TYPE AlbertsSettings EXTENDS TcoData.Entity :
STRUCT
	ServoPosition: REAL;
END_STRUCT
END_TYPE

(* stored: Version 1.1.0.1, ProductVersion 3.1.4024.5
   DUT AlbertsSettings: Id {75fc5a63-d842-05cd-2d7b-d9bf7bef99f3} *)
